Staubli VAL3: Deb2304.pjx

--- Deb2304.pjx ---
Parameters version=s7.4 stackSize=5000 millimeterUnit=true
Program file=Deb2304.pgx
Program file=start.pgx
Program file=stop.pgx
Data file=Deb2304.dtx

--- Deb2304.dtx ---
dio dPowerlinkSorti = {link=POWERLINK-1\%Q0}
mdesc mNomSpeed
mdesc mlent = {accel=9, vel=30, decel=9, blend=off}
tool tstylo = {z=100, fatherId=flange[0], ioLink=valve1}
jointRx ja[5]
  [0] = {j1=-141.592538, j2=84.02454, j3=39.666751, j4=0.388019, j5=55.73836, j6=91.723919}
  [1] = {j1=-141.797065, j2=55.548957, j3=26.304021, j4=0.325386, j5=97.577607, j6=91.780733}
  [2] = {j1=-1.061441, j2=69.857939, j3=0.585564, j4=-0.646318, j5=109.792733, j6=232.256985}
  [3] = {j1=-1.782017, j2=63.511465, j3=34.980386, j4=-0.618292, j5=81.739303, j6=231.843932}
  [4] = {j1=-1.782031, j2=69.640192, j3=39.18089, j4=-0.645507, j5=71.410438, j6=231.960844}
num nPowerlink

--- main.pgx ---
program main()
begin
  while true
    doECAT1_0 = true

    if(diECAT1_0 == true)

      doECAT1_0 = false

      x[0] = diECAT1_1
      x[1] = diECAT1_2
      x[2] = diECAT1_3
      x[3] = diECAT1_4
      x[4] = diECAT1_5
      x[5] = diECAT1_6
      x[6] = diECAT1_7
      x[7] = diECAT1_8

      co_x = x[0] * 1 + x[1] * 2 + x[2] * 4 + x[3] * 8 + x[4] * 16 + x[5] * 32 + x[6] * 64 + x[7] * 128

      y[0] = diECAT1_9
      y[1] = diECAT1_10
      y[2] = diECAT1_11
      y[3] = diECAT1_12
      y[4] = diECAT1_13
      y[5] = diECAT1_14
      y[6] = diECAT1_15
      y[7] = diECAT1_16

      co_y = y[0] * 1 + y[1] * 2 + y[2] * 4 + y[3] * 8 + y[4] * 16 + y[5] * 32 + y[6] * 64 + y[7] * 128


      doECAT1_0 = true

    endIf
  endWhile
end

--- start.pgx ---
program start()
begin
  call Deb2304()
end

--- Deb2304.pgx ---
program Deb2304()
begin

  dPowerlinkSorti[0]=true

  waitEndMove()
  movej(ja[0],tstylo,mlent)
  waitEndMove()
  movej(ja[1],tstylo,mlent)
  waitEndMove()
  movej(ja[2],tstylo,mlent)
  waitEndMove()
  movej(ja[3],tstylo,mlent)
  waitEndMove()
  movej(ja[4],tstylo,mlent)
  waitEndMove()
  movej(ja[3],tstylo,mlent)
  waitEndMove()
  movej(ja[2],tstylo,mlent)
  waitEndMove()
  movej(ja[0],tstylo,mlent)
  waitEndMove()

  dPowerlinkSorti[0]=false
end
